TYPE ST_RecipeInfo :
STRUCT
	sUserCreated		:STRING;
	sUserEdited			:STRING;
	sUserVerified		:STRING;
	sTimeCreated		:STRING;
	sTimeEdited			:STRING;
	sTimeVerified		:STRING;
	bVerification		:BOOL;
	iVersion			:INT;
END_STRUCT
END_TYPE

(* stored: Version 1.1.0.1, ProductVersion 3.1.4026.13
   DUT ST_RecipeInfo: Id {92c46135-3ebd-4abe-9be7-d30ff114d1d9} *)
